PROGRAM SchreibeSollwerte
VAR
END_VAR

CASE SM.Status OF
	
	Lesen:
	
	
	Schreiben:
	
	//Stellsignal Veflüssiger Ventilator
		Soll_VF_Ventilator.INT_VAR_Output:=	FB_Nativ_zu_SPS_lin(output:=Soll_VF_Ventilator);

	//Stellsignal Kompressor
		Soll_KP.INT_VAR_Output:= 			FB_Nativ_zu_SPS_lin(output:=Soll_KP);
	
	//Stellsignal elektrische Heizung
		Soll_ElektHeizrack1.INT_VAR_Output		:= FB_Nativ_zu_SPS_lin(output:= Soll_ElektHeizrack1);
		Soll_ElektHeizrack2.INT_VAR_Output		:= FB_Nativ_zu_SPS_lin(output:= Soll_ElektHeizrack2);
		Soll_ElektHeizrack_Boden.INT_VAR_Output := FB_Nativ_zu_SPS_lin(output:= Soll_ElektHeizrack_Boden);
		
END_CASE

END_PROGRAM

(* stored: Version 1.1.0.1, ProductVersion 3.1.4019.2
   POU SchreibeSollwerte: Id {22df7958-a872-4ced-8935-f8d6650b596d}, SpecialFunc None *)
